(* IEC 61131-3 sources: CodesysTest/alpha/export/FBs/Components/FunnelFB.pou/ClosingTime.prop, 1 file *)

(* ---- Get.pm.st ---- *)
(*#-#-#-#-#-#-#-#-#-#---Declaration---#-#-#-#-#-#-#-#-#-#-#-#-#*)

VAR
END_VAR
(*#-#-#-#-#-#-#-#-#-#---Implementation---#-#-#-#-#-#-#-#-#-#-#-#-#*)

ClosingTime := TO_REAL(closingTimer.PT) / 1000;
